INTERFACE I_FalliblePublic EXTENDS I_Fallible


METHOD ClearError
END_METHOD


METHOD SetError
VAR_INPUT
    sMsg : T_MaxString;
END_VAR
END_METHOD

END_INTERFACE

(* stored: Version 1.1.0.1
   Itf I_FalliblePublic: Id {89b23eb2-9e8f-4419-acc0-6743009400bd}
   Method ClearError: Id {7a06bc68-b3cc-4d54-b1d6-37d3b5bac468}
   Method SetError: Id {49397cf3-2cc3-4d58-bdc0-973ef16a8d2b} *)
